TYPE "OP_PB"
VERSION : 0.1
// Block: OP_PB
   STRUCT
      Rest : Bool;
      Work : Bool;
   END_STRUCT;

END_TYPE
